// TIA Portal V20 export
ORGANIZATION_BLOCK "Main"   // OB1046, LAD, ProgramCycle
TITLE = "Main Program Sweep (Cycle)"
// stored: AutoNumber false, IsIECCheckEnabled true, Namespace Unit1.Em8, SetENOAutomatically true
   VAR_INPUT
      Initial_Call : Bool;   // Initial call of this OB
      Remanence : Bool;   // =True, if remanent data are available
   END_VAR
   VAR_TEMP
      tempIndex : Int;   // Index of EM in the array
   END_VAR
BEGIN

REGION Network 1: Simulation
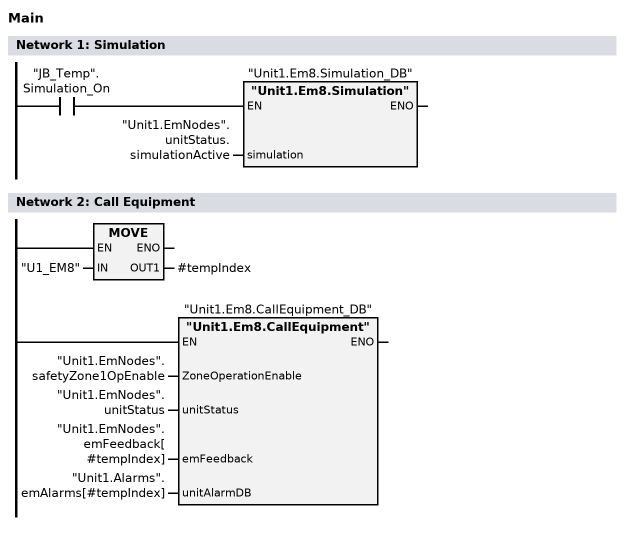
   RUNG wire#powerrail
      Contact( "JB_Temp".Simulation_On )
      "Unit1.Em8.Simulation_DB"(simulation := "Unit1.EmNodes".unitStatus.simulationActive)
   END_RUNG
   // the same network as SCL:
   IF "JB_Temp".Simulation_On THEN
       "Unit1.Em8.Simulation_DB"(simulation := "Unit1.EmNodes".unitStatus.simulationActive);   // "Unit1.Em8.Simulation"
   END_IF;
END_REGION

REGION Network 2: Call Equipment
   RUNG wire#powerrail
      Move(in := "U1_EM8", out1 => #tempIndex)
   END_RUNG
   RUNG wire#powerrail
      "Unit1.Em8.CallEquipment_DB"(ZoneOperationEnable := "Unit1.EmNodes".safetyZone1OpEnable, unitStatus := "Unit1.EmNodes".unitStatus, emFeedback := "Unit1.EmNodes".emFeedback[#tempIndex], unitAlarmDB := "Unit1.Alarms".emAlarms[#tempIndex])
   END_RUNG
   // the same network as SCL:
   #tempIndex := "U1_EM8";
   "Unit1.Em8.CallEquipment_DB"(ZoneOperationEnable := "Unit1.EmNodes".safetyZone1OpEnable,   // "Unit1.Em8.CallEquipment"
                           unitStatus := "Unit1.EmNodes".unitStatus,
                           emFeedback := "Unit1.EmNodes".emFeedback[#tempIndex],
                           unitAlarmDB := "Unit1.Alarms".emAlarms[#tempIndex]);
END_REGION
END_ORGANIZATION_BLOCK
